// Author: Feijian Ni
// Date: 2023.11.22
FUNCTION_BLOCK FB_RedunJntControl_ver2
VAR_INPUT
END_VAR
VAR_OUTPUT
END_VAR
VAR
	// joint 6 deviation from center
	m_jnt6Bias :LREAL;
	
	// max target position step 
	m_maxTargetPosStep :LREAL :=10*g_deg2rad;
	
	// static velocity threshold
	m_staticVelThres :LREAL := 60 *g_deg2Rad;
	
	// static threshold of joint bias
	m_staticBiasThres :LREAL := 30 *g_deg2Rad;
	
	// rudundancy track flag
	m_trackFlag :BOOL;
	
	// joint4 track tolerance
	m_joint4TrackTol :LREAL :=1*g_deg2rad;
	
	// orientation nullspace jacobian
	m_oriNullJaco: Mat4d;
	
	// current manipulation velocity
	m_curManipWVel :LREAL :=0;
	
	// joint4 limit buffer
	m_jntLimitBuffer : LREAL :=2.5*g_deg2Rad;
	
	// control paramters for redundant joint4 position control
//	m_redunJntKp: LREAL:=8.0;
//	m_redunJntKd:LREAL:=0.2;
//	m_redunJntKp: LREAL:=3.0;
//	m_redunJntKd:LREAL:=0.1;
	m_redunJntKp: LREAL:=2.5;
	m_redunJntKd:LREAL:=0.05;
	m_redunJntKi:LREAL:=0;
	m_redunJntKiLimit: LREAL:=200;
	m_redunJntCtrlLimit:LREAL:=1000;

	// max vel and acc for joint4 motion
	m_jnt4MaxFollowVel :LREAL :=2*pi;
	m_jnt4MaxFollowAcc :LREAL :=4*pi;
	m_jnt4MinFollowAcc :LREAL :=1.5*pi;
	m_jnt4MinAccVel:LREAL:= 60 *g_deg2Rad;
	m_jnt4MaxAccVel:LREAL:= 150 *g_deg2Rad;
	
	// max acc scale when approaching joint limit
	m_accScaleNearLimit :LREAL;
	m_maxAccScaleNearLimit :LREAL := 1.0;
	m_accScaleBiasLB :LREAL := 30 *g_deg2Rad;
	m_accScaleBiasUB :LREAL := 45 *g_deg2Rad;

	// final target position of joint4 in motor (not DH , same for below defination) 
	m_jnt4TargetPos: LREAL;
	
	// OTG for joint4 motion
	m_trajFilter :FB_secOrdTrajFilter;
	
	// command joint4 position and veloicty in motor for next cycle
	m_cmdJntPos: LREAL;
	m_cmdJntVel: LREAL;
	m_cmdJntAcc: LREAL;

	// PID for joint position
	m_jntPIDCtrl: FB_PID;
	m_jntCtrlTrq: LREAL;
	
END_VAR

METHOD PROTECTED calcJnt6Bias : LREAL
VAR_IN_OUT CONSTANT
	i_masterArm :FB_MasterArm;
END_VAR
IF 1= i_masterArm.armIdx THEN
	calcJnt6Bias :=i_masterArm.curJntPos[6]+PI/2;
ELSE 
	calcJnt6Bias := i_masterArm.curJntPos[6]-PI/2;
END_IF
END_METHOD

// calculate orientation manipulation velocity(in local coordinate)
METHOD calcManipVel : LREAL
VAR_IN_OUT CONSTANT
	i_masterArm :FB_MasterArm;
END_VAR
VAR
	wVelWrd,wVelLocal:Vec3d;
	rotT:Mat3d;
END_VAR
wVelWrd[1]:= i_masterArm.m_curCartLinkTwist[4];
wVelWrd[2]:= i_masterArm.m_curCartLinkTwist[5];
wVelWrd[3]:= i_masterArm.m_curCartLinkTwist[6];

matTranspose(i_masterArm.curCartPose.m_rot, rotT);
matMultiVec(rotT, wVelWrd, wVelLocal);

wVelLocal[3]:=0;
calcManipVel:=norm(wVelLocal);
END_METHOD

METHOD PROTECTED calcNullJaco : Mat4d;
VAR_IN_OUT CONSTANT
	i_masterArm :FB_MasterArm;
END_VAR
VAR
	i,j:INT;
	oriJaco:Mat34;
	oriJt:Mat43;
	oriJJt:Mat3d;
	oriJJtInv:Mat3d;
	oriJPinv:Mat43;
	JpinvJ :Mat4d;
	eye4d :Mat4d := g_eye4d;
END_VAR
// compute pinv of orientation jacobian
FOR i:=1 TO 3 DO
	FOR j:=1 TO 4 DO
		oriJaco[i,j]:=i_masterArm.simJaco[i+3,j+3];
	END_FOR
END_FOR
matTranspose(oriJaco, oriJt);
matMultiply(oriJaco ,oriJt , oriJJt);
invMat3(oriJJt, oriJJtInv);
matMultiply(oriJt, oriJJtInv, oriJPinv);

// calculate nullspace
matMultiply(oriJPinv, oriJaco, JpinvJ);
matSub(eye4d , JpinvJ, calcNullJaco);
END_METHOD

METHOD PROTECTED calcRedunPos : BOOL
VAR_IN_OUT CONSTANT
	i_masterArm :FB_MasterArm;
END_VAR

VAR 
	j6Bias :LREAL;
	curJntPos : Vec7d;
	jnt4LinkPos, jnt4TargetLinkPos :LREAL;
	singScale:LREAL;
END_VAR
// compute desired joint4 link position
// therotically should be link position, but joint controller use motor pos, so here also use motor pos, or will cause other problems
curJntPos :=  i_masterArm.curJntPos;
jnt4LinkPos:=i_masterArm.jnt4MotorToLink(curJntPos[2],curJntPos[3],curJntPos[4]);

// scale track motion near redundant singularity
IF ABS(m_oriNullJaco[1,1])<g_smallNum THEN
	singScale :=0;
ELSE
	singScale := MAX(ABS(m_oriNullJaco[2,1]/m_oriNullJaco[1,1]), ABS(m_oriNullJaco[3,1]/m_oriNullJaco[1,1]));
END_IF
j6Bias := m_jnt6Bias * ABS(singScale);

j6Bias := LIMIT (-m_maxTargetPosStep, j6Bias, m_maxTargetPosStep);
// final target position
jnt4TargetLinkPos := LIMIT(GVL_ArmJointParameters.g_minJntPos[i_masterArm.armIdx,4]+m_jntLimitBuffer, 
			jnt4LinkPos-j6Bias,GVL_ArmJointParameters.g_maxJntPos[i_masterArm.armIdx,4]-m_jntLimitBuffer); 
			
// convert from link position to motor position
m_jnt4TargetPos:=i_masterArm.jnt4LinkToMotor(curJntPos[2], curJntPos[3], jnt4TargetLinkPos);
END_METHOD

METHOD init : BOOL
VAR_IN_OUT CONSTANT
	i_masterArm :FB_MasterArm;
END_VAR
VAR
	currentRatioMotor2Jnt:LREAL;
END_VAR
m_cmdJntPos:=i_masterArm.curJntPos[4];
m_jnt4TargetPos:=m_cmdJntPos;
m_cmdJntVel:=0;

// init controller
currentRatioMotor2Jnt:=GVL_ArmJointParameters.g_motorTrqConst[4]*GVL_ArmJointParameters.g_motorReduction[4]/1000;
m_jntPIDCtrl.init(g_armCtrlCycleTime,m_redunJntKp,m_redunJntKd,m_redunJntKi,
		m_redunJntKiLimit* currentRatioMotor2Jnt,	m_redunJntCtrlLimit*currentRatioMotor2Jnt);

// init OTG
m_trajFilter.init(m_cmdJntPos,m_cmdJntVel,m_jnt4MaxFollowVel,m_jnt4MaxFollowAcc,g_armCtrlCycleTime);
END_METHOD

METHOD run : LREAL
VAR_IN_OUT CONSTANT
	i_masterArm :FB_MasterArm;
END_VAR
VAR_INPUT
	i_followEnable :BOOL;
END_VAR


VAR
	velScale,limitScale:LREAL;
	maxAcc, minDec:LREAL;
	wVel:Vec3d;

END_VAR
// joint 6 deviation from center
m_jnt6Bias := calcJnt6Bias(i_masterArm);

// calculate nullspace jacobian
m_oriNullJaco := calcNullJaco(i_masterArm);

// calculate manipulation angular velocity(exclude roll velocity)
m_curManipWVel := calcManipVel(i_masterArm);

// check if arm is static
m_trackFlag := startTrackCheck(i_masterArm);

// determin target position of joint4
IF i_followEnable THEN
	// update target redundant joint position
	IF  m_trackFlag THEN
		calcRedunPos(i_masterArm);
	ELSE
		// no control in static state
		IF ABS(m_cmdJntPos-m_jnt4TargetPos)< m_joint4TrackTol THEN
			m_jnt4TargetPos := i_masterArm.curJntPos[4];
			m_cmdJntPos :=i_masterArm.curJntPos[4];
			m_cmdJntVel:=0;
			m_jntPIDCtrl.reset();
			m_trajFilter.init(m_cmdJntPos,m_cmdJntVel,m_jnt4MaxFollowVel,m_jnt4MaxFollowAcc,g_armCtrlCycleTime);
		END_IF
	END_IF
END_IF

// scale following acceleration based on manipulation velocity
velScale := LIMIT (0,(ABS(m_curManipWVel)-m_jnt4MinAccVel)/(m_jnt4MaxAccVel-m_jnt4MinAccVel), 1.0);
maxAcc:=(m_jnt4MaxFollowAcc-m_jnt4MinFollowAcc)*velScale+m_jnt4MinFollowAcc;
//minDec:=m_trajFilter.minDec(m_jnt4TargetPos);
//maxAcc := MAX(maxAcc, minDec);

// scale acceleration when approaching limit
//m_accScaleNearLimit:=1;
limitScale := LIMIT(0.0,(ABS(m_jnt6Bias) - m_accScaleBiasLB)/(m_accScaleBiasUB-m_accScaleBiasLB),1.0);
m_accScaleNearLimit := 1+ limitScale * velScale * m_maxAccScaleNearLimit;
maxAcc:=maxAcc*m_accScaleNearLimit;


// run OTG
m_trajFilter.maxV:=m_curManipWVel;
m_trajFilter.maxA:=maxAcc;
m_trajFilter.run(m_jnt4TargetPos, 0.0, o_cmdAcc=>m_cmdJntAcc,o_cmdVel=>m_cmdJntVel, o_cmdPos=>m_cmdJntPos);

// joint position control torque control
m_jntCtrlTrq:=m_jntPIDCtrl.run(m_cmdJntPos,i_masterArm.curJntPos[4], m_cmdJntVel, i_masterArm.curJntVel[4]);

run:=m_jntCtrlTrq;
END_METHOD

METHOD startTrackCheck : BOOL
VAR_IN_OUT CONSTANT
	i_masterArm :FB_MasterArm;
END_VAR
IF (m_curManipWVel> m_staticVelThres AND i_masterArm.m_curLinkVel[6] * m_jnt6Bias > 0)  OR ABS(m_jnt6Bias)> m_staticBiasThres THEN
	startTrackCheck := TRUE;
ELSE
	startTrackCheck :=FALSE;
END_IF
END_METHOD

END_FUNCTION_BLOCK

(* stored: Version 1.1.0.1, ProductVersion 3.1.4024.11
   POU FB_RedunJntControl_ver2: Id {5e3b737e-31d3-4d77-9e77-17103a194492}, SpecialFunc None
   Method calcJnt6Bias: Id {62da1175-4dee-4a2d-99d7-a2216f69e0c0}
   Method calcManipVel: Id {d30dc0a0-4e04-499e-b7a2-27cbdac68846}
   Method calcNullJaco: Id {44ffb8cc-8ed9-463b-9f14-ab4c68d22fa3}
   Method calcRedunPos: Id {f3d36eb4-ddf4-4ca7-a786-b6dc940eeca2}
   Method init: Id {d697c275-6d85-49d3-be29-358a6bf61d38}
   Method run: Id {4c968ae7-5d7f-496e-9de7-5b02c86d53c0}
   Method startTrackCheck: Id {d9ebb5b9-dcb3-4729-be7a-1fa562b50232} *)
